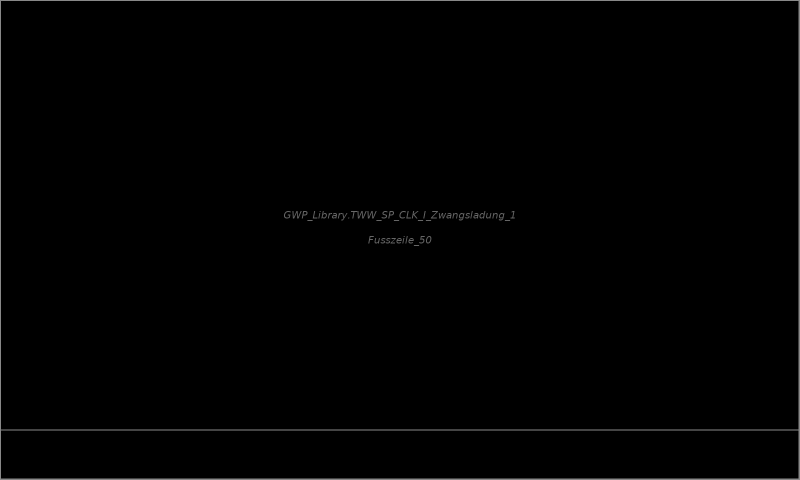
VISUALIZATION TWW_SP_CLK_I_Zwangsladung_1  // 800x480
    Frame (0,0 800x430)
        shows GWP_Library.TWW_SP_CLK_I_Zwangsladung_1(FB_CLK_I := Main.TWW_SP_0.CLK_I_0)
    Frame (0,0 800x480)
        shows Fusszeile_50()
END_VISUALIZATION

(* stored: Version 1.1.0.1, ProductVersion 3.1.4022.6
   Visu TWW_SP_CLK_I_Zwangsladung_1: Id {2e3f04d0-048b-4c1f-81d2-bd7f0b9efc5d} *)
